//冷压工位
PROGRAM LateBlanking_Auto2
VAR
	
	FB_CSP_Velo_Torque_Cold: FB_CSP_Velo_Torque;
	Dne: BOOL;
	SingleStep_2 : R_TRIG;
	TestLengya: R_TRIG;
	b_Cold_TON :ARRAY[1..10] OF ton;
	Sampling_0: Sampling;
	Sampling0: Sampling;
	BBB: BOOL;
	BlowTime:TON;
	BlowCloseTime:TON;
	rt: R_TRIG;
END_VAR

Cold_Press();

  Coldbusy:= FB_CSP_Velo_Torque_Cold.Busy;

b_Cold_TON[2](PT:=T#300MS);
//清零自动复位
b_Cold_TON[1](IN:=Press_Clear[1],PT:=T#300MS);
IF b_Cold_TON[1].Q THEN
	Press_Clear[1]:=FALSE;
END_IF

IF Permit_Blow[1] AND P3_SystemRUN.iMode=1 AND
   LREAL_TO_REAL(arrAxisCtrl[P3AxisNo.P3M1_ColdpreActuated].Status.fActPos) <= arrAxisPar[P3AxisNo.P3M1_ColdpreActuated].arrTargetPoint[4] AND
   LREAL_TO_REAL(arrAxisCtrl[P3AxisNo.P3M1_ColdpreActuated].Status.fActPos) > arrAxisPar[P3AxisNo.P3M1_ColdpreActuated].arrTargetPoint[5] THEN
   arrCyCtrl[P3CYNo.P3ColdBlow].Cmd.bON:=TRUE;//冷压吹气允许信号，冷压驱动当前位置<=吹气开始位且大于吹气结束位,则开始吹气
   arrCyCtrl[P3CYNo.P3ColdBlow].Cmd.bOFF:=FALSE;  
END_IF   


IF  P3_SystemRUN.iMode=1 AND 
    LREAL_TO_REAL(arrAxisCtrl[P3AxisNo.P3M1_ColdpreActuated].Status.fActPos) <= arrAxisPar[P3AxisNo.P3M1_ColdpreActuated].arrTargetPoint[5] THEN
   arrCyCtrl[P3CYNo.P3ColdBlow].Cmd.bON:=FALSE;
   arrCyCtrl[P3CYNo.P3ColdBlow].Cmd.bOFF:=TRUE;//冷压驱动当前位置<=吹气结束位，则吹气关闭
END_IF   

(*BlowTime(IN:=Permit_Blow[1], PT:=T#0S , Q=> , ET=> );
BlowCloseTime(IN:=arrCyCtrl[P3CYNo.P3ColdBlow].Cmd.bON, PT:=T#2S , Q=> , ET=> );
IF BlowTime.Q  THEN//冷压吹气
	arrCyCtrl[P3CYNo.P3ColdBlow].Cmd.bON:=TRUE;
	arrCyCtrl[P3CYNo.P3ColdBlow].Cmd.bOFF:=FALSE;
ELSIF BlowCloseTime.Q  THEN
	arrCyCtrl[P3CYNo.P3ColdBlow].Cmd.bON:=FALSE;
	arrCyCtrl[P3CYNo.P3ColdBlow].Cmd.bOFF:=TRUE;
END_IF*)

FB_CSP_Velo_Torque_Cold.Hold_Time:=P3Par.P3_Press_Time[1]*1000;

P3Senser.P3_Cold_clear:=Press_Clear[1];
SingleStep_2 (CLK:=P3_Start[2] , Q=>);
TestLengya (CLK:=Testone , Q=>);
IF  SingleStep_2.Q  or NOT StepModel[2] THEN
	SingleStep[2]:=FALSE;
END_IF
IF  TestLengya.Q  THEN
	CellMemory[CellNo.Coldpress].Cell:=TRUE;
	Permit_Cold_Press:=TRUE;
	CellMemory[CellNo.Coldpress].Hough:=1;
END_IF

IF P3_SystemRUN.iMode=1  AND LateBlanking_init_OK[2]  THEN
CASE Step31 OF
1://轴和气缸回初始状态
IF NOT SingleStep[2] THEN
	
	arrCyCtrl[P3CYNo.P3ColdPressTensed].Cmd.bON:=TRUE;//冷压麦拉膜气缸松开
	
	IF  (NOT arrAxisCtrl[P3AxisNo.P3M1_ColdpreActuated].Cmd.arrbRealPoint[1]) AND (NOT arrAxisCtrl[P3AxisNo.P3M1_ColdpreActuated].Status.Error) AND arrAxisCtrl[P3AxisNo.P3M1_ColdpreActuated].Status.Homed 
		AND arrAxisCtrl[P3AxisNo.P3M1_ColdpreActuated].Status.Enabled AND arrAxisCtrl[P3AxisNo.P3M1_ColdpreActuated].Status.NoMoving THEN
		arrAxisCtrl[P3AxisNo.P3M1_ColdpreActuated].Cmd.iGoSetPos:=1;	//P3_M1冷压驱动电机去初始位
	END_IF
	
	IF  (NOT arrAxisCtrl[P3AxisNo.P3M1_ColdpreSupPlateLine].Cmd.arrbRealPoint[1]) AND (NOT arrAxisCtrl[P3AxisNo.P3M1_ColdpreSupPlateLine].Status.Error) AND arrAxisCtrl[P3AxisNo.P3M1_ColdpreSupPlateLine].Status.Homed 
		AND arrAxisCtrl[P3AxisNo.P3M1_ColdpreSupPlateLine].Status.Enabled AND arrAxisCtrl[P3AxisNo.P3M1_ColdpreSupPlateLine].Status.NoMoving THEN
		arrAxisCtrl[P3AxisNo.P3M1_ColdpreSupPlateLine].Cmd.iGoSetPos:=1;	//P3_M1冷压麦拉膜电机去初始位
	END_IF
	
	IF  arrAxisCtrl[P3AxisNo.P3M1_ColdpreActuated].Cmd.arrbRealPoint[1] AND arrAxisCtrl[P3AxisNo.P3M1_ColdpreActuated].Status.NoMoving AND arrAxisCtrl[P3AxisNo.P3M1_ColdpreSupPlateLine].Cmd.arrbRealPoint[1] 
		AND arrAxisCtrl[P3AxisNo.P3M1_ColdpreSupPlateLine].Status.NoMoving (*AND arrCyCtrl[P3CYNo.P3ColdPressTensed].Status.OFFState AND NOT arrCyCtrl[P3CYNo.P3ColdPressTensed].Status.Error2*) THEN
		IF  StepModel[2] THEN
			SingleStep[2]:=TRUE;
		ELSE
			SingleStep[2]:=FALSE;
		END_IF		
	Step31:=5;	
	END_IF
	END_IF

	
5:
Step31:=10;
(*	IF NOT P3User2_Par.Shield[7] AND  CellMemory[CellNo.Coldpress].Cell THEN
				Step31:=10;	//如果冷压有电芯记忆则跳至10步
	ELSIF PermitColdPressRack AND arrAxisCtrl[P3AxisNo.P3M1_ColdpreActuated].Cmd.arrbRealPoint[1]  AND P3User2_Par.Shield[7]
				AND arrAxisCtrl[P3AxisNo.P3M1_ColdpreActuated].Status.Homed AND  arrAxisCtrl[P3AxisNo.P3M1_ColdpreActuated].Status.NoMoving
				AND NOT CellMemory[CellNo.Coldpress].Cell AND arrAxisCtrl[P3AxisNo.P3M1_ColdpreSupPlateLine].Cmd.arrbRealPoint[1]
				AND arrAxisCtrl[P3AxisNo.P3M1_ColdpreSupPlateLine].Status.Homed  AND  arrAxisCtrl[P3AxisNo.P3M1_ColdpreSupPlateLine].Status.NoMoving THEN	
					Step31:=7;//如果有允许冷压上料信号,冷压驱动在初始位,没有冷压电芯记忆,冷压托板开合在初始位，则跳至7步
	END_IF


7://如果烤箱上料夹进退在初始位，烤箱上料夹搬运当前位置大于其冷压位,冷压上料夹进退在初始位,冷压上料夹平移当前位置>=其初始位,则冷压托板开合去张开位
IF NOT SingleStep[2] THEN
    arrCyCtrl[P3CYNo.P3ColdPressTensed].Cmd.bON:=TRUE;//冷压麦拉膜气缸张紧
	IF  (arrAxisCtrlV2[P3AxisNo.P3_M2_OvenRetracting].Cmd.arrbRealPoint[43] OR LREAL_TO_REAL(arrAxisCtrlV2[P3AxisNo.P3_M2_OvenCarrying].Status.fActPos)>arrAxisParV2[P3AxisNo.P3_M2_OvenCarrying].arrTargetPoint[44]) AND 
       	(arrAxisCtrl[P3AxisNo.P3M1_ColdpreRetracting].Cmd.arrbRealPoint[1] OR LREAL_TO_REAL(arrAxisCtrl[P3AxisNo.P3M1_ColdpreLine].Status.fActPos)>=arrAxisPar[P3AxisNo.P3M1_ColdpreLine].arrTargetPoint[1]) AND 
      	 (NOT arrAxisCtrl[P3AxisNo.P3M1_ColdpreSupPlateLine].Cmd.arrbRealPoint[2]) AND (NOT arrAxisCtrl[P3AxisNo.P3M1_ColdpreSupPlateLine].Status.Error) AND arrAxisCtrl[P3AxisNo.P3M1_ColdpreSupPlateLine].Status.Homed 
		AND arrAxisCtrl[P3AxisNo.P3M1_ColdpreSupPlateLine].Status.Enabled AND arrAxisCtrl[P3AxisNo.P3M1_ColdpreSupPlateLine].Status.NoMoving THEN
		arrAxisCtrl[P3AxisNo.P3M1_ColdpreSupPlateLine].Cmd.iGoSetPos:=2;	//P3_M1冷压麦拉膜电机去张开位
	END_IF
	
	IF  arrAxisCtrl[P3AxisNo.P3M1_ColdpreSupPlateLine].Cmd.arrbRealPoint[2] AND arrAxisCtrl[P3AxisNo.P3M1_ColdpreSupPlateLine].Status.NoMoving  THEN
		IF  StepModel[2] THEN
			SingleStep[2]:=TRUE;
		ELSE
			SingleStep[2]:=FALSE;
		END_IF
	Step31:=8;	
	END_IF
	END_IF


8://如果有冷压允许上料信号、冷压驱动在初始位\贴胶下料在3055步、没有冷压电芯记忆、冷压上料夹进退在冷压位,则跳至9步
	IF  PermitColdPressRack AND arrAxisCtrl[P3AxisNo.P3M1_ColdpreActuated].Cmd.arrbRealPoint[1] AND Step30=3055
		AND arrAxisCtrl[P3AxisNo.P3M1_ColdpreActuated].Status.Homed AND  arrAxisCtrl[P3AxisNo.P3M1_ColdpreActuated].Status.NoMoving
		AND NOT CellMemory[CellNo.Coldpress].Cell AND arrAxisCtrl[P3AxisNo.P3M1_ColdpreRetracting].Cmd.arrbRealPoint[5] 
		AND arrAxisCtrl[P3AxisNo.P3M1_ColdpreRetracting].Status.NoMoving AND arrAxisCtrl[P3AxisNo.P3M1_ColdpreRetracting].Status.Homed THEN
			Step31:=9;	
	END_IF
	
9://冷压托板开合到初始位
IF NOT SingleStep[2] THEN
	IF  (NOT arrAxisCtrl[P3AxisNo.P3M1_ColdpreSupPlateLine].Cmd.arrbRealPoint[1]) AND (NOT arrAxisCtrl[P3AxisNo.P3M1_ColdpreSupPlateLine].Status.Error) AND arrAxisCtrl[P3AxisNo.P3M1_ColdpreSupPlateLine].Status.Homed 
		AND arrAxisCtrl[P3AxisNo.P3M1_ColdpreSupPlateLine].Status.Enabled AND arrAxisCtrl[P3AxisNo.P3M1_ColdpreSupPlateLine].Status.NoMoving THEN
		arrAxisCtrl[P3AxisNo.P3M1_ColdpreSupPlateLine].Cmd.iGoSetPos:=1;	//P3_M1冷压麦拉膜电机去初始位
	END_IF
	
	IF  arrAxisCtrl[P3AxisNo.P3M1_ColdpreActuated].Cmd.arrbRealPoint[1] AND arrAxisCtrl[P3AxisNo.P3M1_ColdpreActuated].Status.NoMoving 
		AND arrAxisCtrl[P3AxisNo.P3M1_ColdpreSupPlateLine].Cmd.arrbRealPoint[1] AND arrAxisCtrl[P3AxisNo.P3M1_ColdpreSupPlateLine].Status.NoMoving  THEN
		IF  StepModel[2] THEN
			SingleStep[2]:=TRUE;
		ELSE
			SingleStep[2]:=FALSE;
		END_IF	
		Step31:=10;
	END_IF
END_IF	
	*)
10://如果有允许冷压信号、冷压驱动在初始位、冷压有电芯记忆、没有冷压完成信号、冷压托板开合在初始位，则跳至15步
IF NOT SingleStep[2] THEN
IF  Permit_Cold_Press AND arrAxisCtrl[P3AxisNo.P3M1_ColdpreActuated].Cmd.arrbRealPoint[1] 
	AND CellMemory[CellNo.Coldpress].Cell AND NOT Cold_Press_Finish 
	AND arrAxisCtrl[P3AxisNo.P3M1_ColdpreSupPlateLine].Cmd.arrbRealPoint[1] THEN
	Step31:=15;
	ColdPress_start:=FALSE;
	 Press_Clear[1]:=TRUE;		
		IF  StepModel[2] THEN
				SingleStep[2]:=TRUE;
			ELSE
				SingleStep[2]:=FALSE;
		END_IF
END_IF
END_IF

15://冷压压力上下限为设定压力+-150
CellMemory[CellNo.Coldpress].ColdPress_SV:=P3Par.P3_Press_SV[1];
CellMemory[CellNo.Coldpress].ColdPress_SV_H:=P3Par.P3_Press_SV[1]+150;
CellMemory[CellNo.Coldpress].ColdPress_SV_L:=P3Par.P3_Press_SV[1]-150;
CellMemory[CellNo.Coldpress].ColdPress_Time:=TIME_TO_UINT(P3Par.P3_Press_Time[1]);
CellMemory[CellNo.Coldpress].ColdPress_PVTime:=TIME_TO_UINT(P3Par.P3_Press_Time[1]);
Step31:=20;	


20://如果烤箱上料夹进退在初始位、烤箱上料夹搬运当前位置大于其冷压位、冷压上料夹进退在初始位、冷压上料夹平移当前位置>=其初始位，则冷压托板开合去张开位
IF NOT SingleStep[2] THEN
    arrCyCtrl[P3CYNo.P3ColdPressTensed].Cmd.bON:=TRUE;//冷压麦拉膜气缸张紧
	
	IF  (arrAxisCtrlV2[P3AxisNo.P3_M2_OvenRetracting].Cmd.arrbRealPoint[43] OR LREAL_TO_REAL(arrAxisCtrlV2[P3AxisNo.P3_M2_OvenCarrying].Status.fActPos)>arrAxisParV2[P3AxisNo.P3_M2_OvenCarrying].arrTargetPoint[44]) AND 
       	(arrAxisCtrl[P3AxisNo.P3M1_ColdpreRetracting].Cmd.arrbRealPoint[1] OR LREAL_TO_REAL(arrAxisCtrl[P3AxisNo.P3M1_ColdpreLine].Status.fActPos)>=arrAxisPar[P3AxisNo.P3M1_ColdpreLine].arrTargetPoint[1]) AND 
      	 (NOT arrAxisCtrl[P3AxisNo.P3M1_ColdpreSupPlateLine].Cmd.arrbRealPoint[2]) AND (NOT arrAxisCtrl[P3AxisNo.P3M1_ColdpreSupPlateLine].Status.Error) AND arrAxisCtrl[P3AxisNo.P3M1_ColdpreSupPlateLine].Status.Homed 
		AND arrAxisCtrl[P3AxisNo.P3M1_ColdpreSupPlateLine].Status.Enabled AND arrAxisCtrl[P3AxisNo.P3M1_ColdpreSupPlateLine].Status.NoMoving THEN
		arrAxisCtrl[P3AxisNo.P3M1_ColdpreSupPlateLine].Cmd.iGoSetPos:=2;	//P3_M1冷压麦拉膜电机去张开位
	END_IF
	
	IF  arrAxisCtrl[P3AxisNo.P3M1_ColdpreSupPlateLine].Cmd.arrbRealPoint[2] AND arrAxisCtrl[P3AxisNo.P3M1_ColdpreSupPlateLine].Status.NoMoving 
		AND (*arrCyCtrl[P3CYNo.P3ColdPressTensed].Status.ONState AND *)   NOT arrCyCtrl[P3CYNo.P3ColdPressTensed].Status.Error2 THEN
		IF  StepModel[2] THEN
			SingleStep[2]:=TRUE;
		ELSE
			SingleStep[2]:=FALSE;
		END_IF
	ColdPress_start:=FALSE;
	Step31:=30;	
	END_IF
	END_IF

30://如果烤箱上料夹进退在初始位、烤箱上料夹搬运当前位置>=其冷压位,烤箱上料夹进退在初始位、烤箱上料夹平移当前位置>=其初始位、冷压托板开合在张开位,有允许冷压信号、下料安全条件、冷压电芯记忆，则冷压开始
arrCyCtrl[P3CYNo.P3ColdPressTensed].Cmd.bON:=TRUE;//冷压麦拉膜气缸张紧
IF  (arrAxisCtrlV2[P3AxisNo.P3_M2_OvenRetracting].Cmd.arrbRealPoint[43] OR LREAL_TO_REAL(arrAxisCtrlV2[P3AxisNo.P3_M2_OvenCarrying].Status.fActPos)>arrAxisParV2[P3AxisNo.P3_M2_OvenCarrying].arrTargetPoint[44]) AND 
    (arrAxisCtrl[P3AxisNo.P3M1_ColdpreRetracting].Cmd.arrbRealPoint[1] OR LREAL_TO_REAL(arrAxisCtrl[P3AxisNo.P3M1_ColdpreLine].Status.fActPos)>=arrAxisPar[P3AxisNo.P3M1_ColdpreLine].arrTargetPoint[1]) AND 
	arrAxisCtrl[P3AxisNo.P3M1_ColdpreSupPlateLine].Cmd.arrbRealPoint[2] AND arrAxisCtrl[P3AxisNo.P3M1_ColdpreSupPlateLine].Status.NoMoving 
	 AND Permit_Cold_Press AND b_Press_condition[1] AND CellMemory[CellNo.Coldpress].Cell THEN
	ColdPress_start:=TRUE;
	Sampling_finish[1]:=FALSE;
	Step31:=35;
ELSIF NOT b_Press_condition[1] THEN
	P3_Error[62]:=TRUE;//冷压空压报警
END_IF




50://轴和气缸回初始状态
IF NOT SingleStep[2] THEN
	
	arrCyCtrl[P3CYNo.P3ColdPressTensed].Cmd.bON:=TRUE;//冷压麦拉膜气缸
	
	IF  (NOT arrAxisCtrl[P3AxisNo.P3M1_ColdpreActuated].Cmd.arrbRealPoint[1]) AND (NOT arrAxisCtrl[P3AxisNo.P3M1_ColdpreActuated].Status.Error) AND arrAxisCtrl[P3AxisNo.P3M1_ColdpreActuated].Status.Homed 
		AND arrAxisCtrl[P3AxisNo.P3M1_ColdpreActuated].Status.Enabled AND arrAxisCtrl[P3AxisNo.P3M1_ColdpreActuated].Status.NoMoving THEN
		arrAxisCtrl[P3AxisNo.P3M1_ColdpreActuated].Cmd.iGoSetPos:=1;	//P3_M1冷压驱动电机去初始位
	END_IF
	
	IF  (NOT arrAxisCtrl[P3AxisNo.P3M1_ColdpreSupPlateLine].Cmd.arrbRealPoint[1]) AND (NOT arrAxisCtrl[P3AxisNo.P3M1_ColdpreSupPlateLine].Status.Error) AND arrAxisCtrl[P3AxisNo.P3M1_ColdpreSupPlateLine].Status.Homed 
		AND arrAxisCtrl[P3AxisNo.P3M1_ColdpreSupPlateLine].Status.Enabled AND arrAxisCtrl[P3AxisNo.P3M1_ColdpreSupPlateLine].Status.NoMoving THEN
		arrAxisCtrl[P3AxisNo.P3M1_ColdpreSupPlateLine].Cmd.iGoSetPos:=1;	//P3_M1冷压麦拉膜电机去初始位
	END_IF
	
	IF  arrAxisCtrl[P3AxisNo.P3M1_ColdpreActuated].Cmd.arrbRealPoint[1] AND arrAxisCtrl[P3AxisNo.P3M1_ColdpreActuated].Status.NoMoving AND arrAxisCtrl[P3AxisNo.P3M1_ColdpreSupPlateLine].Cmd.arrbRealPoint[1] 
		AND arrAxisCtrl[P3AxisNo.P3M1_ColdpreSupPlateLine].Status.NoMoving (*AND arrCyCtrl[P3CYNo.P3ColdPressTensed].Status.ONState AND NOT arrCyCtrl[P3CYNo.P3ColdPressTensed].Status.Error1  *) THEN
		IF  StepModel[2] THEN
			SingleStep[2]:=TRUE;
		ELSE
			SingleStep[2]:=FALSE;
		END_IF	
Permit_Cold_Press :=FALSE;
Cold_Press_Finish:=TRUE;	
	Step31:=1;	
	END_IF
	END_IF




 
END_CASE
END_IF








IF P3_SystemRUN.iMode=1 OR P3_SystemRUN.iMode=3 THEN
CASE Step31 OF
35://采集完成，冷压实际压力等于采集平均压力值
IF Sampling_finish[1] THEN
CellMemory[CellNo.Coldpress].ColdPress_PV:=Sampling_mean[1]; 
//CellMemory[CellNo.Coldpress].HeatActPos:=LREAL_TO_REAL(arrAxisCtrlV2[P3AxisNo.P3M1_ColdpreActuated].Status.fActPos);
   Step31:=40;	
 END_IF  
40:
b_Cold_TON[2].IN:=TRUE;
IF FB_CSP_Velo_Torque_Cold.HoldOK  AND  FB_CSP_Velo_Torque_Cold.Done AND b_Cold_TON[2].Q THEN
b_Cold_TON[2].IN:=FALSE;
 ColdPress_start:=FALSE;
 Step31:=50;	
END_IF 


END_CASE
END_IF


rt (CLK:=Pressing[1] , Q=>);
IF rt .Q THEN
	CellMemory[CellNo.Coldpress].coldActPos:=LREAL_TO_REAL(arrAxisCtrl[P3AxisNo.P3M1_ColdpreActuated].Status.fActPos);
END_IF

ACTION Cold_Press:
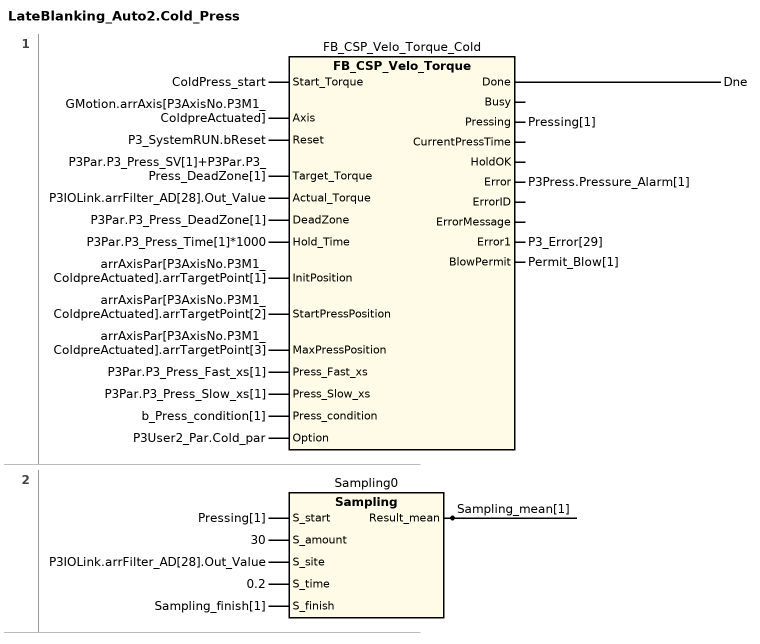
// NETWORK 1
FB_CSP_Velo_Torque_Cold(
    Start_Torque := ColdPress_start,
    Axis := GMotion.arrAxis[P3AxisNo.P3M1_ColdpreActuated],
    Reset := P3_SystemRUN.bReset,
    Target_Torque := P3Par.P3_Press_SV[1]+P3Par.P3_Press_DeadZone[1],
    Actual_Torque := P3IOLink.arrFilter_AD[28].Out_Value,
    DeadZone := P3Par.P3_Press_DeadZone[1],
    Hold_Time := P3Par.P3_Press_Time[1]*1000,
    InitPosition := arrAxisPar[P3AxisNo.P3M1_ColdpreActuated].arrTargetPoint[1],
    StartPressPosition := arrAxisPar[P3AxisNo.P3M1_ColdpreActuated].arrTargetPoint[2],
    MaxPressPosition := arrAxisPar[P3AxisNo.P3M1_ColdpreActuated].arrTargetPoint[3],
    Press_Fast_xs := P3Par.P3_Press_Fast_xs[1],
    Press_Slow_xs := P3Par.P3_Press_Slow_xs[1],
    Press_condition := b_Press_condition[1],
    Option := P3User2_Par.Cold_par,
    Pressing => Pressing[1],
    Error => P3Press.Pressure_Alarm[1],
    Error1 => P3_Error[29],
    BlowPermit => Permit_Blow[1]); // FB_CSP_Velo_Torque
Dne := FB_CSP_Velo_Torque_Cold.Done;

// NETWORK 2
Sampling0(
    S_start := Pressing[1],
    S_amount := 30,
    S_site := P3IOLink.arrFilter_AD[28].Out_Value,
    S_time := 0.2,
    S_finish := Sampling_finish[1],
    Result_mean => Sampling_mean[1]); // Sampling
END_ACTION

END_PROGRAM

(* stored: Version 1.1.0.1, ProductVersion 3.1.4024.12
   POU LateBlanking_Auto2: Id {07baaf96-13b7-4517-89a6-6b359d1104f2}, SpecialFunc None
   Action Cold_Press: Id {dfceb768-4c79-43aa-8499-475372b8e91e} *)
